TYPE ST_BaseDefinition :
STRUCT
	Name		: STRING(40);
	Station		: string(40);
END_STRUCT
END_TYPE

(* stored: Version 1.1.0.1
   DUT ST_BaseDefinition: Id {55ecabba-df22-47a7-bcdf-fa724bff02cb} *)
